// TIA Portal V19 export
FUNCTION "FC_TEST" : Void   // FC123, LAD
   VAR_TEMP
      tVar1 : USInt;
      tVar2 : UInt;
   END_VAR
BEGIN

REGION Network 1
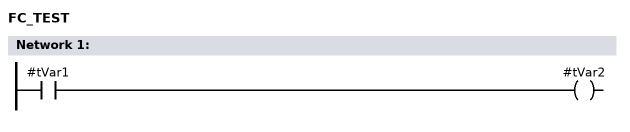
   RUNG wire#powerrail
      Contact( #tVar1 )
      Coil( #tVar2 )
   END_RUNG
   // the same network as SCL:
   #tVar2 := #tVar1;
END_REGION
END_FUNCTION
